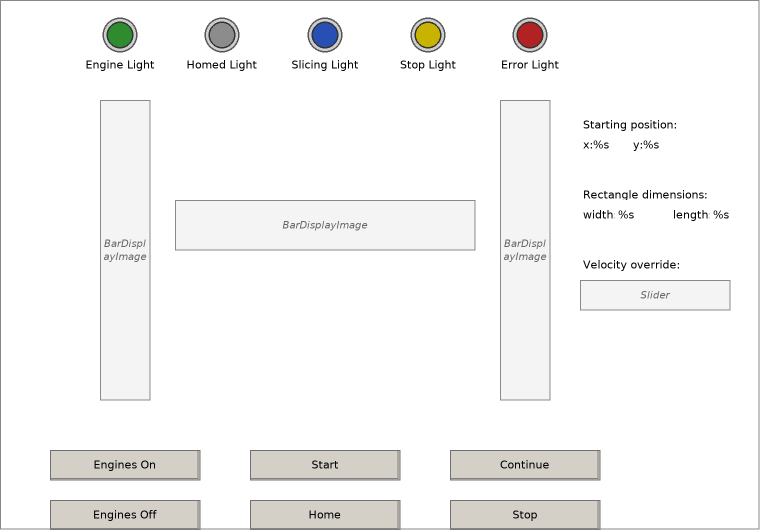
VISUALIZATION Visualization  // 760x530
    Button (250,450 150x30), "Start"
        tap MAIN.bStartButton
    BarDisplayImage (100,100 50x300), value: MAIN.fbSlicer.AxisM1.NcToPlc.ActPos, style: BarDisplayImage-Gray, scale format: %.1f, scale 0..100
    BarDisplayImage (500,100 50x300), value: MAIN.fbSlicer.AxisM1s.NcToPlc.ActPos, style: BarDisplayImage-Gray, scale format: %.1f, scale 0..100
    BarDisplayImage (175,200 300x50), value: MAIN.fbSlicer.AxisM2.NcToPlc.ActPos, style: BarDisplayImage-Gray, scale format: %.1f, scale 0..100
    Button (450,500 150x30), "Stop"
        tap MAIN.bStopButton
    Button (50,450 150x30), "Engines On"
        tap MAIN.bEnginesOnButton
    Button (50,500 150x30), "Engines Off"
        tap MAIN.bEnginesOffButton
    Button (250,500 150x30), "Home"
        tap MAIN.bHomeButton
    Lamp1 (100,15 40x40), variable: MAIN.bEnginesLight, style: Lamp-Lamp1-Green
    Lamp1 (202,15 40x40), variable: MAIN.bHomedLight, style: Lamp-Lamp1-Gray
    Lamp1 (305,15 40x40), variable: MAIN.bSlicingLight, style: Lamp-Lamp1-Blue
    Lamp1 (510,15 40x40), variable: MAIN.bErrorLight, style: Lamp-Lamp1-Red
    Label (80,50 80x30), "Engine Light"
    Label (182,50 80x30), "Homed Light"
    Label (285,50 80x30), "Slicing Light"
    Label (490,50 80x30), "Error Light"
    Rectangle (590,130 50x30), "%s", text variable: MAIN.aStartingPosition[0]
        OnMouseClick: write MAIN.aStartingPosition[0] via Default
    Label (580,110 150x30), "Starting position:"
    Rectangle (640,130 50x30), "%s", text variable: MAIN.aStartingPosition[1]
        OnMouseClick: write MAIN.aStartingPosition[1] via Default
    Label (580,180 150x30), "Rectangle dimensions:"
    Button (450,450 150x30), "Continue"
        tap MAIN.bContinueButton
    Lamp1 (408,15 40x40), variable: MAIN.bStopLight, style: Lamp-Lamp1-Yellow
    Label (388,50 80x30), "Stop Light"
    Slider (580,280 150x30), variable: MAIN.fVelocityOverride, scale 0..100
    Label (580,250 150x30), "Velocity override:"
    Label (580,130 20x30), "x:"
    Label (630,130 20x30), "y:"
    Label (580,200 50x30), "width:"
    Label (670,200 50x30), "length:"
    Rectangle (710,200 50x30), "%s", text variable: MAIN.aSlicingDimensions[1]
        OnMouseClick: write MAIN.aSlicingDimensions[1] via Default
    Rectangle (615,200 50x30), "%s", text variable: MAIN.aSlicingDimensions[0]
        OnMouseClick: write MAIN.aSlicingDimensions[0] via Default
END_VISUALIZATION

(* stored: Version 1.1.0.1, ProductVersion 3.1.4024.12
   Visu Visualization: Id {dfe7afd8-adb6-4863-9d8e-f039d2d76741} *)
